{attribute addProperty BoxType "AX8118-0000-0102-0102"}
{attribute addProperty Id "DeviceDevice_F82A60211620Ch_ACh_A_B17182A2176220WcStateAT %I*WcState_98A4DF7520.250InfoDataAT %I*InfoData_F030DC9B200250"}
{attribute addProperty CRC "3898025815"}
{attribute addProperty SizeInBites "394"}
{attribute addProperty SizeInBytes "49.25"}
TYPE AX8118_2B905711 :
STRUCT
	{attribute addProperty Name "Device"}
	Device : Device_F82A6021;
	{attribute addProperty Name "Ch_A"}
	Ch_A : Ch_A_B17182A2;
	{attribute addProperty Name "WcState"}
	WcState : WcState_98A4DF75;
	{attribute addProperty Name "InfoData"}
	InfoData : InfoData_F030DC9B;
END_STRUCT
END_TYPE

(* stored: Version 1.2.0.0, ProductVersion 3.1.4024.9
   DUT AX8118_2B905711: Id {3ad01ddf-f7b0-45cd-8ee4-687e206f4cd1} *)
